FUNCTION "FC_Separator" : Void
{ S7_Optimized_Access := 'TRUE' }
VERSION : 0.3
   VAR_IN_OUT
      S : "UDT_Separator";
      B : "UDT_BaseMechanism";
   END_VAR

   VAR_TEMP
      elapsedMs : DInt;
      nowTck : DInt;
      forceBreaker : Bool;
      forceFeedback : Bool;
      forceStopTimeout : Bool;
      isFault : Bool;
      isBlocked : Bool;
   END_VAR


BEGIN

	REGION "0) Декодування форсування"
	    // BIT8(256)=forceFeedback, BIT6(64)=forceStopTimeout
	    #forceFeedback := (#B.Force_Code AND 256) <> 0;
	    #forceStopTimeout := (#B.Force_Code AND 64) <> 0;
	END_REGION

	REGION "1) RESET (Тільки за умови усунення причини)"
	    IF #B.Cmd = "CMD_RESET" THEN
	        IF (#B.FLTCode AND "FLT_NO_FEEDBACK") <> 0 THEN
	            IF #S.DI_Feedback_OK OR #forceFeedback THEN
	                #B.FLTCode := #B.FLTCode AND NOT "FLT_NO_FEEDBACK";
	            END_IF;
	        END_IF;
	        IF (#B.FLTCode AND "FLT_STOP_TIMEOUT") <> 0 THEN
	            IF NOT #S.DI_Feedback_OK OR #forceStopTimeout THEN
	                #B.FLTCode := #B.FLTCode AND NOT "FLT_STOP_TIMEOUT";
	            END_IF;
	        END_IF;

	        IF #B.FLTCode = "FLT_NONE" AND #B.Status = "STS_FAULT" THEN
	            #B.Status := "STS_IDLE";
	            #S.StartMs := 0;
	            #S.FeedbackLostMs := 0;
	            #S.StopMs := 0;
	        END_IF;
	    END_IF;
	END_REGION

	REGION "2) Обробка блокувань"
	    IF NOT #B.Enable_OK THEN
	        #B.Status := "STS_DISABLED";
	        #isBlocked := TRUE;
	    ELSIF #B.LocalManual THEN
	        #B.Status := "STS_LOCAL";
	        #isBlocked := TRUE;
	    ELSE
	        #isBlocked := FALSE;
	        IF (#B.Status = "STS_DISABLED") OR (#B.Status = "STS_LOCAL") THEN
	            #B.Status := "STS_IDLE";
	        END_IF;
	    END_IF;
	END_REGION

	REGION "3) Моніторинг аварій (Diagnostic Latch)"
	    // DI_Breaker_OK не використовується для Separator
	END_REGION

	REGION "4) Визначення виконавчої аварії"
	    #isFault := FALSE;
	    IF #B.FLTCode <> "FLT_NONE" THEN
	        IF (#B.FLTCode AND "FLT_NO_FEEDBACK") <> 0 AND NOT #forceFeedback THEN
	            #isFault := TRUE;
	        END_IF;
	        IF (#B.FLTCode AND "FLT_STOP_TIMEOUT") <> 0 AND NOT #forceStopTimeout THEN
	            #isFault := TRUE;
	        END_IF;
	    END_IF;

	    IF #isFault THEN
	        #B.Status := "STS_FAULT";
	    END_IF;
	    #isFault := (#B.Status = "STS_FAULT");
	END_REGION

	REGION "5 & 6) Машина станів та виконання команд"
	    IF (NOT #isFault) AND (NOT #isBlocked) THEN
	        IF #B.Cmd <> "CMD_NONE" THEN
	            #B.LastCmd := #B.Cmd;
	        END_IF;

	        CASE #B.Status OF
	            "STS_IDLE":
	                IF #B.Cmd = "CMD_START" THEN
	                    // Перевірка мінімального інтервалу перезапуску
	                    IF #S.LastStopMs = 0 OR "FC_TimeElapsedMs"(StartTck := #S.LastStopMs, TimeoutMs := "TimeoutMs_Separator_MinRestart",
	                                                                ElapsedMs => #elapsedMs, NowTck => #nowTck) THEN
	                        #B.Status := "STS_STARTING";
	                        #S.StartMs := TIME_TCK();
	                    END_IF;
	                END_IF;

	            "STS_STARTING":
	                IF #S.DI_Feedback_OK OR #forceFeedback THEN
	                    #B.Status := "STS_RUNNING";
	                ELSE
	                    IF "FC_TimeElapsedMs"(StartTck := #S.StartMs, TimeoutMs := "TimeoutMs_Separator_Feedback",
	                                              ElapsedMs => #elapsedMs, NowTck => #nowTck) THEN
	                        #B.FLTCode := #B.FLTCode OR "FLT_NO_FEEDBACK";
	                        #B.Status := "STS_FAULT";
	                    END_IF;
	                END_IF;

	            "STS_RUNNING":
	                IF NOT (#S.DI_Feedback_OK OR #forceFeedback) THEN
	                    IF #S.FeedbackLostMs = 0 THEN
	                        #S.FeedbackLostMs := TIME_TCK();
	                    END_IF;
	                    IF "FC_TimeElapsedMs"(StartTck := #S.FeedbackLostMs, TimeoutMs := "TimeoutMs_Separator_FeedbackPause",
	                                              ElapsedMs => #elapsedMs, NowTck => #nowTck) THEN
	                        #B.FLTCode := #B.FLTCode OR "FLT_NO_FEEDBACK";
	                        #B.Status := "STS_FAULT";
	                    END_IF;
	                ELSE
	                    #S.FeedbackLostMs := 0;
	                END_IF;

	            "STS_STOPPING":
	                IF (NOT #S.DI_Feedback_OK) OR #forceFeedback THEN
	                    #B.Status := "STS_IDLE";
	                    #S.StopMs := 0;
	                    #S.LastStopMs := TIME_TCK();  // Зберігаємо час останньої зупинки
	                ELSE
	                    IF #S.StopMs = 0 THEN
	                        #S.StopMs := TIME_TCK();
	                    END_IF;
	                    IF "FC_TimeElapsedMs"(StartTck := #S.StopMs, TimeoutMs := "TimeoutMs_Separator_Stop",
	                                              ElapsedMs => #elapsedMs, NowTck => #nowTck) THEN
	                        #B.FLTCode := #B.FLTCode OR "FLT_STOP_TIMEOUT";
	                        #B.Status := "STS_FAULT";
	                    END_IF;
	                END_IF;
	        END_CASE;

	        IF #B.Cmd = "CMD_STOP" AND #B.Status <> "STS_IDLE" THEN
	            IF #B.Status = "STS_STARTING" THEN
	                #S.StartMs := 0;
	            END_IF;
	            #B.Status := "STS_STOPPING";
	            #S.StopMs := 0;
	        END_IF;
	    END_IF;
	END_REGION

	REGION "7) Фіналізація"
	    #S.DO_Run := (#B.Status = "STS_STARTING") OR (#B.Status = "STS_RUNNING");
	    #B.Cmd := "CMD_NONE";
	END_REGION

END_FUNCTION
